// TIA Portal project "Automatic Pumping and Draining" (V17)
// Automatic Pumping and Draining
// When Start Pushbutton is pressed and released, then the pump should run for 20s to fill the tank and then drain valve should open for 10s to drain the tank.
// When Stop Pushbutton is pressed and released, the system will stop immediately.

(* hardware
DEVICE "S7-1200 station_1"  S7-1200 Station
   slot 0: "Rack_0"  S7-1200 Rack  Rack  V1.0
   slot 1: "PLC_1"  CPU 1212C AC/DC/Rly  6ES7 212-1BE40-0XB0  V4.5
*)

// ===== PLC "PLC_1"  CPU 1212C AC/DC/Rly =====

VAR_GLOBAL   // PLC tag table "Default tag table"
   "PB_start" AT %I0.0 : Bool;
   "PB_stop" AT %I0.1 : Bool;
   "Pump" AT %Q0.0 : Bool;
   "Drain valve" AT %Q0.1 : Bool;
   "Tag_1" AT %M0.0 : Bool;
   "Tag_2" AT %MD0 : Time;
   "Tag_3" AT %MD4 : Time;
END_VAR

// folder: System blocks/Program resources

DATA_BLOCK "IEC_Timer_0_DB"   // DB1
{ S7_Optimized_Access := 'TRUE' }
AUTHOR : Simatic
FAMILY : IEC
NAME : IEC_TMR
VERSION : 1.0
// stored: InstanceOfName IEC_TIMER
"IEC_TIMER"
BEGIN
END_DATA_BLOCK

DATA_BLOCK "IEC_Timer_0_DB_1"   // DB2
{ S7_Optimized_Access := 'TRUE' }
AUTHOR : Simatic
FAMILY : IEC
NAME : IEC_TMR
VERSION : 1.0
// stored: InstanceOfName IEC_TIMER
"IEC_TIMER"
BEGIN
END_DATA_BLOCK

// folder: (top level)

ORGANIZATION_BLOCK "Main"   // OB1, LAD, ProgramCycle
TITLE = "Main Program Sweep (Cycle)"
{ S7_Optimized_Access := 'TRUE' }
VERSION : 0.1
   VAR_INPUT
      Initial_Call : Bool;   // Initial call of this OB
      Remanence : Bool;   // =True, if remanent data are available
   END_VAR
BEGIN

REGION Network 1
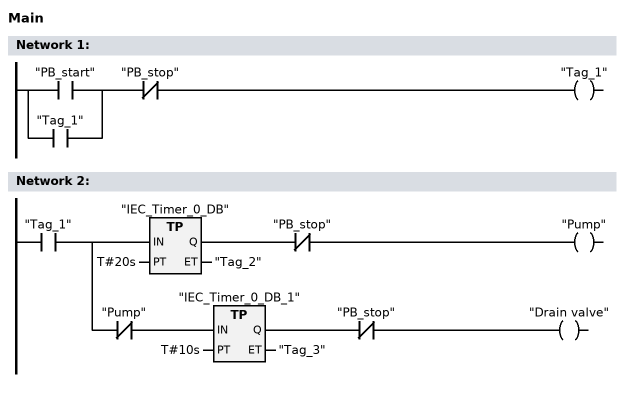
   RUNG wire#powerrail
      Contact( "PB_start" )
      wire#w1
      I_Contact( "PB_stop" )
      Coil( "Tag_1" )
   END_RUNG
   RUNG wire#powerrail
      Contact( "Tag_1" )
   END_RUNG wire#w1
   // the same network as SCL:
   "Tag_1" := ("PB_start" OR "Tag_1") AND NOT "PB_stop";
END_REGION

REGION Network 2
   "IEC_Timer_0_DB".TP(IN := "Tag_1", PT := T#20s, ET => "Tag_2");
   "Pump" := "IEC_Timer_0_DB".Q AND NOT "PB_stop";
   "IEC_Timer_0_DB_1".TP(IN := "Tag_1" AND NOT "Pump", PT := T#10s, ET => "Tag_3");
   "Drain valve" := "IEC_Timer_0_DB_1".Q AND NOT "PB_stop";
END_REGION
END_ORGANIZATION_BLOCK